DATA_BLOCK "ID_PE_Plate_Grafcet"
{ S7_Optimized_Access := 'TRUE' }
VERSION : 0.1
NON_RETAIN
"FB_PE_Plate_Rotate"

BEGIN

END_DATA_BLOCK

